				bManInterlockLiftOut := NOT bManualZIsSafe;
				bManInterlockOut := NOT ((aTRobotAxis[LA_Z1].lrCurrentPos < (alrSafePos[LA_Z1]+lrSafeTolerance)) AND (aTRobotAxis[LA_Z2].lrCurrentPos < (alrSafePos[LA_Z2]+lrSafeTolerance)) AND
								 (*(aTRobotAxis[LA_X].lrCurrentPos < (alrSafePos[LA_X]+lrSafeTolerance)) AND (aTRobotAxis[LA_Y].lrCurrentPos < (alrSafePos[LA_Y]+lrSafeTolerance)) AND*)
								(*AND ((aTRobotAxis[LA_Z1].eCurrentState = AS_InPosition) OR (aTRobotAxis[LA_Z1].eCurrentState = AS_PowerOff))
								AND ((aTRobotAxis[LA_Z2].eCurrentState = AS_InPosition)  OR (aTRobotAxis[LA_Z2].eCurrentState = AS_PowerOff))*)
								(*(aTRobotAxis[LA_X].bAxisHomed) AND (aTRobotAxis[LA_Y].bAxisHomed) AND*)
								(aTRobotAxis[LA_Z1].bAxisHomed) AND (aTRobotAxis[LA_Z2].bAxisHomed) AND bPlateTakerIsUp);
				CASE sCurrentState.eStep OF
					SP_ManualStp0 :
						TManualCmd.TPlateVacuum.Enable := TRUE;
						TManualCmd.THead1Vacuum.Enable := TRUE;
						TManualCmd.THead2Vacuum.Enable := TRUE;
						TManualCmd.TPlateVacuum.Activate := bEnablePlateVacuum;
						TManualCmd.TMovePlateTakerDown.Activate := bMovePlateTakerDown;
						TManualCmd.THead1Vacuum.Activate := abEnableHeadVacuum[0];
						TManualCmd.THead2Vacuum.Activate := abEnableHeadVacuum[1];
						FOR iAxis := 0 TO 4 DO
							TManualCmd.aTAxis[iAxis].Home.Activate := FALSE;
							TManualCmd.aTAxis[iAxis].MoveFw.Activate := FALSE;
							TManualCmd.aTAxis[iAxis].MoveBw.Activate := FALSE;
							TManualCmd.aTAxisPos[iAxis].MoveToTeach.Activate := FALSE;
							TManualCmd.aTAxisPos[iAxis].Teach := FALSE;
							TManualCmd.aTAxisPos[iAxis].MoveToTeach.Enable := FALSE;
							TManualCmd.aTAxis[iAxis].JogStep := alrJogStep[iAxis];
						END_FOR
						FOR i:= 0 TO 1 DO
							TManualCmd.alrVaccumThershold[i] := alrVacuumThreshold[i];
						END_FOR
						TManualCmd.TVisionCalibration.Activate := FALSE;
						TManualCmd.TSafe.Activate := FALSE;
						TManualCmd.TZSensorTeach.Activate := FALSE;
						 iManMoveAxis:=iManMoveAxisNone;
						TManualCmd.TAspirationBrush.Enable := TRUE;
						TManualCmd.TAspirationBrush.Activate := bAspirationBrushOn;
						TManualCmd.lrSensorAdjust := lrSensorAdjust;
						TManualCmd.TMoveVision2Table.Activate := FALSE;
						TManualCmd.TMoveVision2Lift.Activate := FALSE;
						sCurrentState.eStep := SP_ManualStp1;
					SP_ManualStp1 :
						IF bStopReq THEN
							sCurrentState.eStatus := MS_Stopped;
						ELSE
							FOR iAxis := 0 TO 4 DO
								iTeachedAxis := GetLoaderTeachedAxisFromAxis(iAxis);
								IF TManualCmd.aTAxisPos[iAxis].Teach THEN
									TManualCmd.aTAxisPos[iAxis].Teach := FALSE; (* change here the learning teach *)
									IF (iRobotOffset = LTO_Z1) THEN
										alrRobotOffset[iTeachedAxis,iRobotOffset] := 0;
										alrRobotPos[iTeachedAxis, iRobotPosition] := aTRobotAxis[iAxis].lrCurrentPos;
										iTeachedModeDebug := 0;
									ELSIF (iRobotOffset <> LTO_Plate) THEN (* Plate position are hardcoded, cannot be teached *)
										alrRobotOffset[iTeachedAxis, iRobotOffset] := aTRobotAxis[iAxis].lrCurrentPos - alrRobotPos[iTeachedAxis, iRobotPosition];
										iTeachedModeDebug := 1;
									END_IF
								END_IF
								IF (alrJogStep[iAxis] <> TManualCmd.aTAxis[iAxis].JogStep) THEN
									alrJogStep[iAxis] := TManualCmd.aTAxis[iAxis].JogStep;
								END_IF
								IF TManualCmd.aTAxisPos[iAxis].MoveToTeach.Activate AND iManMoveAxis=iManMoveAxisNone THEN
									alrTargetPos[iAxis] := TManualCmd.aTAxisPos[iAxis].TeachedPos;
									iManMoveAxis := iAxis;
									sCurrentState.eStep := SP_ManualStp10;
								END_IF
								IF TManualCmd.aTAxis[iAxis].MoveFw.Activate AND iManMoveAxis=iManMoveAxisNone THEN
									alrTargetPos[iAxis] := aTRobotAxis[iAxis].lrCurrentPos + alrJogStep[iAxis];
									iManMoveAxis := iAxis;
									sCurrentState.eStep := SP_ManualStp10;
								END_IF
								IF TManualCmd.aTAxis[iAxis].MoveBw.Activate AND iManMoveAxis=iManMoveAxisNone THEN
									alrTargetPos[iAxis] := aTRobotAxis[iAxis].lrCurrentPos - alrJogStep[iAxis];
									iManMoveAxis := iAxis;
									sCurrentState.eStep := SP_ManualStp10;
								END_IF
								IF TManualCmd.aTAxis[iAxis].Home.Activate AND  iManMoveAxis=iManMoveAxisNone THEN
									iManMoveAxis := iAxis;
									sCurrentState.eStep := SP_ManualStp20;
								END_IF
							END_FOR
							FOR i:= 0 TO 1 DO
								IF TManualCmd.alrVaccumThershold[i] <> alrVacuumThreshold[i] THEN
									alrVacuumThreshold[i] := TManualCmd.alrVaccumThershold[i];
								END_IF
							END_FOR
							IF TManualCmd.TSafe.Activate AND  iManMoveAxis=iManMoveAxisNone THEN
								TManualCmd.TSafe.Activate := FALSE;
								iManMoveAxis:=LA_X;
								sCurrentState.eStep := SP_ManualStp30;
							END_IF
							IF TManualCmd.TVisionCalibration.Activate AND  iManMoveAxis=iManMoveAxisNone THEN
								TManualCmd.TVisionCalibration.Activate := FALSE;
								iManMoveAxis:=LA_X;
								sCurrentState.eStep := SP_ManualStp50;
							END_IF
							IF (lrSensorAdjust <> TManualCmd.lrSensorAdjust) THEN
								lrSensorAdjust :=  TManualCmd.lrSensorAdjust;
							END_IF
							IF TManualCmd.TZSensorTeach.Activate THEN
								TManualCmd.TZSensorTeach.Activate := FALSE;
								lrSensorAdjust := 0 - (TSensorMeasure.lrValue - lrSensorAdjust);
								TManualCmd.lrSensorAdjust := lrSensorAdjust;
							END_IF
							IF TManualCmd.TMoveVision2Table.Activate  AND  iManMoveAxis=iManMoveAxisNone THEN
								TManualCmd.TMoveVision2Table.Activate := FALSE;
								iManMoveAxis:=LA_X;
								alrTargetPos[LA_X] := alrRobotPos[LTA_X,LTP_TableSideALayering1]  -  sPartDataMMI.alrPartOffsetLayering[sRunData.iLayringOffsetPos].lrX + alrRobotOffset[LTA_X, LTO_Vision];
								alrTargetPos[LA_Y] :=  alrRobotPos[LTA_Y,LTP_TableSideALayering1]  + sPartDataMMI.alrPartOffsetLayering[sRunData.iLayringOffsetPos].lrY + alrRobotOffset[LTA_Y, LTO_Vision];
								sCurrentState.eStep := SP_ManualStp70;
							END_IF
							IF TManualCmd.TMoveVision2Lift.Activate  AND  iManMoveAxis=iManMoveAxisNone THEN
								TManualCmd.TMoveVision2Lift.Activate := FALSE;
								iManMoveAxis:=LA_X;
								alrTargetPos[LA_X] := alrRobotPos[LTA_X,LTP_Lift1] + alrRobotOffset[LTA_X, LTO_Vision] + alrLiftCalibrationOffset[LTP_Lift1,LTA_X]  - sPlateData.alrPartOnPlate[TManualCmd.wMoveVision2LiftPos-1].lrX ;
								alrTargetPos[LA_Y] :=  alrRobotPos[LTA_Y,LTP_Lift1] + alrRobotOffset[LTA_Y, LTO_Vision] + alrLiftCalibrationOffset[LTP_Lift1,LTA_Y] - sPlateData.alrPartOnPlate[TManualCmd.wMoveVision2LiftPos-1].lrY ;
								sCurrentState.eStep := SP_ManualStp70;
							END_IF
						END_IF
					SP_ManualStp10: (* Do the movement *)
						aeMoveRobotCommand[iManMoveAxis] := AC_MoveAtAbsPos;
						sCurrentState.eStep := SP_ManualStp11;
					SP_ManualStp11: (* Wait until position is reached *)
						CASE aTRobotAxis[iManMoveAxis].eCurrentState OF
							AS_InPosition, AS_InError:
								FOR iAxis := 0 TO 4 DO
									TManualCmd.aTAxis[iAxis].Home.Activate := FALSE;
									TManualCmd.aTAxis[iAxis].MoveFw.Activate := FALSE;
									TManualCmd.aTAxis[iAxis].MoveBw.Activate := FALSE;
									TManualCmd.aTAxisPos[iAxis].MoveToTeach.Activate := FALSE;
								END_FOR
								 iManMoveAxis:=iManMoveAxisNone;
								sCurrentState.eStep := SP_ManualStp1;
						END_CASE
					SP_ManualStp20 : (* Init axis *)
						aeMoveRobotCommand[iManMoveAxis] := AC_Home;
						sCurrentState.eStep := SP_ManualStp21;
					SP_ManualStp21 : (* Rotate the turn over to go to index position *)
						CASE aTRobotAxis[iManMoveAxis].eCurrentState OF
							AS_InPosition, AS_InError:
								FOR iAxis := 0 TO 4 DO
									TManualCmd.aTAxis[iAxis].Home.Activate := FALSE;
									TManualCmd.aTAxis[iAxis].MoveFw.Activate := FALSE;
									TManualCmd.aTAxis[iAxis].MoveBw.Activate := FALSE;
								END_FOR
								 iManMoveAxis:=iManMoveAxisNone;
								sCurrentState.eStep := SP_ManualStp1;
						END_CASE
					SP_ManualStp30: (* Move taker up *)
						TManualCmd.TMovePlateTakerDown.Activate := FALSE;
						IF bPlateTakerIsUp THEN
							sCurrentState.eStep := SP_ManualStp31;
						ELSIF bJackError THEN
							iManMoveAxis:=iManMoveAxisNone;
							sCurrentState.eStep := SP_ManualStp1;
						END_IF
					SP_ManualStp31: (*Move  Z1 and Z2 to Limit*)
						aeMoveRobotCommand[LA_Z1] := AC_MoveLimitNeg;
						aeMoveRobotCommand[LA_Z2] := AC_MoveLimitNeg;
						sCurrentState.eStep := SP_ManualStp32;
					SP_ManualStp32:
						IF aTRobotAxis[LA_Z1].eCurrentState= AS_OnLimitNeg AND aTRobotAxis[LA_Z2].eCurrentState= AS_OnLimitNeg THEN
							sCurrentState.eStep := SP_ManualStp33;
						ELSIF (aTRobotAxis[LA_Z1].eCurrentState= AS_OnLimitNeg AND aTRobotAxis[LA_Z2].eCurrentState = AS_InError) OR
							    (aTRobotAxis[LA_Z1].eCurrentState= AS_InError AND aTRobotAxis[LA_Z2].eCurrentState = AS_OnLimitNeg) OR
							    (aTRobotAxis[LA_Z1].eCurrentState= AS_InError AND aTRobotAxis[LA_Z2].eCurrentState = AS_InError) THEN
							iManMoveAxis:=iManMoveAxisNone;
							sCurrentState.eStep := SP_ManualStp1;
						END_IF
					SP_ManualStp33: (* Init X/Y  *)
						aeMoveRobotCommand[LA_X] := AC_Init;
						aeMoveRobotCommand[LA_Y] := AC_Init;
						sCurrentState.eStep := SP_ManualStp34;
					SP_ManualStp34:
						IF aTRobotAxis[LA_X].eCurrentState= AS_InPosition AND aTRobotAxis[LA_Y].eCurrentState = AS_InPosition THEN
							sCurrentState.eStep := SP_ManualStp35;
						ELSIF (aTRobotAxis[LA_X].eCurrentState= AS_InPosition AND aTRobotAxis[LA_Y].eCurrentState = AS_InError) OR
							    (aTRobotAxis[LA_X].eCurrentState= AS_InError AND aTRobotAxis[LA_Y].eCurrentState = AS_InPosition) OR
							    (aTRobotAxis[LA_X].eCurrentState= AS_InError AND aTRobotAxis[LA_Y].eCurrentState = AS_InError) THEN
							iManMoveAxis:=iManMoveAxisNone;
							sCurrentState.eStep := SP_ManualStp1;
						END_IF
					SP_ManualStp35: (* Move X/Y *)
						aeMoveRobotCommand[LA_X] := AC_MoveAtAbsPos;
						aeMoveRobotCommand[LA_Y] := AC_MoveAtAbsPos;
						alrTargetPos[LA_X] := alrSafePos[LA_X];
						alrTargetPos[LA_Y] := alrSafePos[LA_Y];
						sCurrentState.eStep := SP_ManualStp36;
					SP_ManualStp36:
						IF aTRobotAxis[LA_X].eCurrentState= AS_InPosition AND aTRobotAxis[LA_Y].eCurrentState = AS_InPosition THEN
							sCurrentState.eStep := SP_ManualStp37;
						ELSIF (aTRobotAxis[LA_X].eCurrentState= AS_InPosition AND aTRobotAxis[LA_Y].eCurrentState = AS_InError) OR
							    (aTRobotAxis[LA_X].eCurrentState= AS_InError AND aTRobotAxis[LA_Y].eCurrentState = AS_InPosition) OR
							    (aTRobotAxis[LA_X].eCurrentState= AS_InError AND aTRobotAxis[LA_Y].eCurrentState = AS_InError) THEN
							iManMoveAxis:=iManMoveAxisNone;
							sCurrentState.eStep := SP_ManualStp1;
						END_IF
					SP_ManualStp37: (* Init Z1 and Z2*)
						aeMoveRobotCommand[LA_Z1] := AC_Init;
						aeMoveRobotCommand[LA_Z2] := AC_Init;
						sCurrentState.eStep := SP_ManualStp38;
					SP_ManualStp38:
						IF aTRobotAxis[LA_Z1].eCurrentState= AS_InPosition AND aTRobotAxis[LA_Z2].eCurrentState = AS_InPosition THEN
							sCurrentState.eStep := SP_ManualStp39;
						ELSIF (aTRobotAxis[LA_Z1].eCurrentState= AS_InPosition AND aTRobotAxis[LA_Z2].eCurrentState = AS_InError) OR
							    (aTRobotAxis[LA_Z1].eCurrentState= AS_InError AND aTRobotAxis[LA_Z2].eCurrentState = AS_InPosition) OR
							    (aTRobotAxis[LA_Z1].eCurrentState= AS_InError AND aTRobotAxis[LA_Z2].eCurrentState = AS_InError) THEN
							iManMoveAxis:=iManMoveAxisNone;
							sCurrentState.eStep := SP_ManualStp1;
						END_IF
					SP_ManualStp39: (* Move up Z1 and Z2 *)
						aeMoveRobotCommand[LA_Z1] := AC_MoveAtAbsPos;
						aeMoveRobotCommand[LA_Z2] := AC_MoveAtAbsPos;
						alrTargetPos[LA_Z1] := alrSafePos[LA_Z1];
						alrTargetPos[LA_Z2] := alrSafePos[LA_Z2];
						sCurrentState.eStep := SP_ManualStp40;
					SP_ManualStp40:
						IF (aTRobotAxis[LA_Z1].eCurrentState= AS_InPosition OR aTRobotAxis[LA_Z1].eCurrentState = AS_InError) AND
							    (aTRobotAxis[LA_Z2].eCurrentState= AS_InPosition OR aTRobotAxis[LA_Z2].eCurrentState = AS_InError) THEN
							iManMoveAxis:=iManMoveAxisNone;
							sCurrentState.eStep := SP_ManualStp1;
						END_IF
					SP_ManualStp50: (*Switch part for learning vision *)
						iHead := 0;
						alrTargetPos[LA_X] := alrRobotPos[LTA_X,LTP_TableSideALayering1] + alrRobotOffset[LTA_X, iHead];
						alrTargetPos[LA_Y] :=  alrRobotPos[LTA_Y,LTP_TableSideALayering1] + alrRobotOffset[LTA_Y, iHead];
						alrTargetPos[LA_THETA] := alrRobotPos[LTA_THETA,LTP_TableSideALayering1] + alrRobotOffset[LTA_THETA, iHead];
						ZPositionTakeGive := alrRobotPos[LTA_Z,LTP_TableSideALayering1] + alrRobotOffset[LTA_Z, iHead];
						alrTargetPos[LA_X] := alrTargetPos[LA_X]   -  sPartDataMMI.alrPartOffsetLayering[0].lrX;
						alrTargetPos[LA_Y] := alrTargetPos[LA_Y]  + sPartDataMMI.alrPartOffsetLayering[0].lrY;
						ZPositionTakeGive := ZPositionTakeGive + (lrCalibrationLayeringAndPartAndHeadHeight - sPartDataMMI.lrLayeringAndPartAndHeadHeight);
						aeMoveRobotCommand[LA_X] := AC_MoveAtAbsPos;
						aeMoveRobotCommand[LA_Y] := AC_MoveAtAbsPos;
						aeMoveRobotCommand[LA_THETA] := AC_MoveAtAbsPos;
						sCurrentState.eStep := SP_ManualStp51;
					SP_ManualStp51:
						IF eRobotXYTStatus = AS_InPosition THEN
							sCurrentState.eStep := SP_ManualStp52;
						END_IF
					SP_ManualStp52 :  (*Take Part*)
						ZPosition := ZPositionTakeGive + sPartDataMMI.lrPartOffsetZLayeringTake;
						alrTargetPos[LA_Z1+iHead] := ZPosition;
						aeMoveRobotCommand[LA_Z1+iHead] := AC_MoveAtAbsPos;
						sCurrentState.eStep := SP_ManualStp53;
					SP_ManualStp53 :  (*Movement done*)
						IF aTRobotAxis[LA_Z1+iHead].lrRemainingTimeToGo < 1 AND aTRobotAxis[LA_Z1+iHead].lrRemainingTimeToGo <> 0 THEN
							 TManualCmd.THead1Vacuum.Activate := TRUE;
						END_IF
						IF aTRobotAxis[LA_Z1+iHead].eCurrentState = AS_InPosition THEN
							 TManualCmd.THead1Vacuum.Activate := TRUE;
							sCurrentState.eStep := SP_ManualStp54;
						END_IF
					SP_ManualStp54 :
						(* Check if the part is on head *)
						IF aTHeadVacuum[iHead].bVacuumCorrect THEN
							alrTargetPos[LA_Z1+iHead] := alrSafePos[LA_Z1+iHead];
							aeMoveRobotCommand[LA_Z1+iHead] := AC_MoveAtAbsPos;
							sCurrentState.eStep := SP_ManualStp55;
						END_IF
					SP_ManualStp55 :  (*Movement done*)
						IF aTRobotAxis[LA_Z1+iHead].eCurrentState = AS_InPosition THEN
							iPlatePos := 0;
							iZSensorPositionScan := 0;
							sCurrentState.eStep := SP_ManualStp56;
						END_IF
					SP_ManualStp56:
						alrTargetPos[LA_X] := alrRobotPos[LTA_X,LTP_Lift2] + alrRobotOffset[LTA_X, LTO_ZSensor] + alrLiftCalibrationOffset[LTP_Lift2,LTA_X]  -  sPlateData.alrPartOnPlate[iPlatePos].lrX - sPartDataMMI.alrSensorZOffset[iZSensorPositionScan].lrX;
						alrTargetPos[LA_Y] :=alrRobotPos[LTA_Y,LTP_Lift2] + alrRobotOffset[LTA_Y, LTO_ZSensor] + alrLiftCalibrationOffset[LTP_Lift2,LTA_Y] - sPlateData.alrPartOnPlate[iPlatePos].lrY - sPartDataMMI.alrSensorZOffset[iZSensorPositionScan].lrY;
						aeMoveRobotCommand[LA_X] := AC_MoveAtAbsPos;
						aeMoveRobotCommand[LA_Y] := AC_MoveAtAbsPos;
						TSensorZWaitStab(IN := FALSE);
						sCurrentState.eStep := SP_ManualStp57;
					SP_ManualStp57:
						IF eRobotXYTStatus = AS_InPosition THEN
							TSensorZWaitStab(IN := TRUE, PT := TSensorZWaitStabTime);
							IF TSensorZWaitStab.Q THEN
								IF TSensorMeasure.bInputOutOfRange THEN
									iManMoveAxis:=iManMoveAxisNone;
									sCurrentState.eStep := SP_ManualStp1;
									bZSensorOutOfRangeError := TRUE;
								END_IF
								lrZSensorPosition[iZSensorPositionScan] := TSensorMeasure.lrValue;
								IF iZSensorPositionScan = 0 AND (sPartDataMMI.alrSensorZOffset[1].lrX<>0 OR sPartDataMMI.alrSensorZOffset[1].lrY<>0) THEN
									iZSensorPositionScan := iZSensorPositionScan + 1;
									sCurrentState.eStep := SP_ManualStp56;
								ELSE
									sCurrentState.eStep := SP_ManualStp58;
								END_IF
							END_IF
						END_IF
					SP_ManualStp58: (* Move to take position *)
						IF iZSensorPositionScan = 1 THEN
							(* We used two position, mean the value *)
							ZPositionTakeGive := (lrZSensorPosition[0] + lrZSensorPosition[1]) / 2;
						ELSE
							(* Only one position, use the first one then *)
							ZPositionTakeGive := lrZSensorPosition[0];
						END_IF
						ZPositionTakeGive := alrRobotPos[LTA_Z,LTP_TableSideALayering1] + alrRobotOffset[LTA_Z, iHead] + (lrCalibrationPartAndHeadHeight - sPartDataMMI.lrPartAndHeadHeight) - ZPositionTakeGive;
						alrTargetPos[LA_X] := alrRobotPos[LTA_X,LTP_Lift2] + alrRobotOffset[LTA_X, iHead] + alrLiftCalibrationOffset[LTP_Lift2,LTA_X]  -  sPlateData.alrPartOnPlate[iPlatePos].lrX;
						alrTargetPos[LA_Y] :=alrRobotPos[LTA_Y,LTP_Lift2] + alrRobotOffset[LTA_Y, iHead] + alrLiftCalibrationOffset[LTP_Lift2,LTA_Y] - sPlateData.alrPartOnPlate[iPlatePos].lrY;
						alrTargetPos[LA_THETA] := alrRobotPos[LTA_THETA,LTP_TableSideALayering1] + alrRobotOffset[LTA_THETA, iHead];
						aeMoveRobotCommand[LA_THETA] := AC_MoveAtAbsPos;
						aeMoveRobotCommand[LA_X] := AC_MoveAtAbsPos;
						aeMoveRobotCommand[LA_Y] := AC_MoveAtAbsPos;
						sCurrentState.eStep := SP_ManualStp59;
					SP_ManualStp59:
						IF eRobotXYTStatus = AS_InPosition THEN
							ZPosition := ZPositionTakeGive + sPartDataMMI.lrPartOffsetZLiftDrop;
							sCurrentState.eStep := SP_ManualStp60;
						END_IF
					SP_ManualStp60 : (*Give Part*)
						alrTargetPos[LA_Z1+iHead] := ZPosition + 1;
						aeMoveRobotCommand[LA_Z1+iHead] := AC_MoveAtAbsPos;
						sCurrentState.eStep := SP_ManualStp61;
					SP_ManualStp61 :  (*Movement done*)
						IF aTRobotAxis[LA_Z1+iHead].eCurrentState = AS_InPosition THEN
							 TManualCmd.THead1Vacuum.Activate := FALSE;
							sCurrentState.eStep := SP_ManualStp62;
						END_IF
					SP_ManualStp62:
						(* Check if laying vacuum is disabled *)
						IF aTHeadVacuum[iHead].bVacuumCorrect THEN
							alrTargetPos[LA_Z1+iHead] := alrSafePos[LA_Z1+iHead];
							aeMoveRobotCommand[LA_Z1+iHead] := AC_MoveAtAbsPos;
							sCurrentState.eStep := SP_ManualStp63;
						END_IF
					SP_ManualStp63 :
						IF aTRobotAxis[LA_Z1+iHead].eCurrentState = AS_InPosition THEN
							alrTargetPos[LA_X] := alrRobotPos[LTA_X,LTP_Lift2] + alrRobotOffset[LTA_X, LTO_Vision] + alrLiftCalibrationOffset[LTP_Lift2,LTA_X]  - sPlateData.alrPartOnPlate[iPlatePos].lrX ;
							alrTargetPos[LA_Y] :=  alrRobotPos[LTA_Y,LTP_Lift2] + alrRobotOffset[LTA_Y, LTO_Vision] + alrLiftCalibrationOffset[LTP_Lift2,LTA_Y] - sPlateData.alrPartOnPlate[iPlatePos].lrY ;
							aeMoveRobotCommand[LA_X] := AC_MoveAtAbsPos;
							aeMoveRobotCommand[LA_Y] := AC_MoveAtAbsPos;
							sCurrentState.eStep := SP_ManualStp64;
						END_IF
					SP_ManualStp64:
						IF eRobotXYTStatus = AS_InPosition THEN
							iManMoveAxis:=iManMoveAxisNone;
							sCurrentState.eStep := SP_ManualStp1;
						END_IF
					SP_ManualStp70: (* Move X/Y *)
						aeMoveRobotCommand[LA_X] := AC_MoveAtAbsPos;
						aeMoveRobotCommand[LA_Y] := AC_MoveAtAbsPos;
						sCurrentState.eStep := SP_ManualStp71;
					SP_ManualStp71:
						IF aTRobotAxis[LA_X].eCurrentState= AS_InPosition AND aTRobotAxis[LA_Y].eCurrentState = AS_InPosition THEN
							iManMoveAxis:=iManMoveAxisNone;
							sCurrentState.eStep := SP_ManualStp1;
						END_IF
				END_CASE
				abEnableHeadVacuum[0] := TManualCmd.THead1Vacuum.Activate;
				abEnableHeadVacuum[1] := TManualCmd.THead2Vacuum.Activate;
				bMovePlateTakerDown := TManualCmd.TMovePlateTakerDown.Activate;
				bEnablePlateVacuum := TManualCmd.TPlateVacuum.Activate;
				TManualCmd.lrSensorAdjust := lrSensorAdjust;
				bAspirationBrushOn := TManualCmd.TAspirationBrush.Activate;
			MS_Paused:
				IF bStopReq THEN
					sCurrentState.eStatus := MS_Ready;
				END_IF
		END_CASE;
	MC_Init :
		sCurrentState.eStep := SP_InitStp1;
		sCurrentState.eStatus := MS_Init;
	MC_Run :
		sCurrentState.eStatus := MS_Running;
	MC_Manual :
		sCurrentState.bInitDone := FALSE;
		sCurrentState.eStatus := MS_Manual;
		sCurrentState.eStep := SP_ManualStp0;
	MC_Stop :
		sCurrentState.eStatus := MS_Stopped;
END_CASE;

IF bResetErrors THEN
	sCurrentState.bInError := FALSE;
	bZSensorOutOfRangeError := FALSE;
END_IF

IF bNewJob THEN
	IF C_PROD_MODE_GOOD_PART THEN
		IF sProdLot.dGoodQty > 0 THEN
			sProdLot.dEstimatedPartTime := TIME_TO_DWORD(TJobElapsed)  / sProdLot.dGoodQty;
		ELSE
			sProdLot.dEstimatedPartTime := 0;
		END_IF
	ELSE
		IF sProdLot.dProdQty > 0 THEN
			sProdLot.dEstimatedPartTime := TIME_TO_DWORD(TJobElapsed)  / sProdLot.dProdQty;
		ELSE
			sProdLot.dEstimatedPartTime := 0;
		END_IF
	END_IF
	sProdLot.dLoadedQty := sProdLot.dProdQty;
END_IF

IF bNewJob THEN
(*IF bNewJob OR sCurrentState.eStatus = MS_Manual THEN*)
	abResetPlateState[LPP_Lift1] := TRUE;
	abResetPlateState[LPP_Lift2] := TRUE;
	abResetPlateState[LPP_Reject] := TRUE;
END_IF
IF bNewPlateLift1 THEN abResetPlateState[LPP_Lift1] := TRUE; END_IF
IF bNewPlateLift2 THEN abResetPlateState[LPP_Lift2] := TRUE; END_IF
IF bNewPlateReject THEN abResetPlateState[LPP_Reject] := TRUE; END_IF

IF abCopySwitchFromPlate THEN
	abCopySwitchFromPlate := FALSE;
	FOR j := 0 TO sPlateData.iNbPartOnPlate DO
		aTPartOnSwitchPlate[j].ePartStatus := aTPartOnPlate[LPP_Lift1, j].ePartStatus;
	END_FOR
END_IF

FOR i :=LPP_Reject  TO LPP_Lift2 DO
	IF abResetPlateState[i] THEN
		abResetPlateState[i] := FALSE;
		FOR j := 0 TO sPlateData.iNbPartOnPlate DO
			aTPartOnPlate[i, j ].ePartStatus := PPS_Undefined;
		END_FOR
	END_IF
END_FOR

IF abCopySwitchToPlate THEN
	abCopySwitchToPlate := FALSE;
	FOR j := 0 TO sPlateData.iNbPartOnPlate DO
		aTPartOnPlate[LPP_Lift2, j].ePartStatus := aTPartOnSwitchPlate[j].ePartStatus;
	END_FOR
END_IF
(* ----------------------------------------------------------- MOVE SECURITY CHECK -------------------------------------------------------------------------*)

(* Check if a consequent move more then 2 mm with heads down or plate taker down is requested *)
IF ((ABS(aTRobotAxis[LA_X].lrCurrentPos - alrTargetPos[LA_X]) > lrMaxXYMoveAllowed) AND (aeMoveRobotCommand[LA_X] <> AC_None)) OR
		((ABS(aTRobotAxis[LA_Y].lrCurrentPos - alrTargetPos[LA_Y]) > lrMaxXYMoveAllowed) AND (aeMoveRobotCommand[LA_Y] <> AC_None)) THEN
	IF (aTRobotAxis[LA_Z1].lrCurrentPos > (alrSecuredSafeZPos[0] + lrSafeTolerance))
			OR (aTRobotAxis[LA_Z2].lrCurrentPos > (alrSecuredSafeZPos[1] + lrSafeTolerance))
			OR NOT bPlateTakerIsUp THEN
		IF sCurrentState.eStep <> SP_RunStp63 THEN (* Do not check during cleaning *)
			aeMoveRobotCommand[LA_X] := AC_ForceStop;
			aeMoveRobotCommand[LA_Y] := AC_ForceStop;
			aeMoveRobotCommand[LA_Z1] := AC_ForceStop;
			aeMoveRobotCommand[LA_Z2] := AC_ForceStop;
			sCurrentState.bInitDone := FALSE;
			bConflictDetected := TRUE;
		END_IF
	END_IF
ELSIF ((aTRobotAxis[LA_X].lrCurrentPos > alrUnsecuredArea[0,LA_X]+ lrSafeTolerance) AND (aTRobotAxis[LA_X].lrCurrentPos < alrUnsecuredArea[1,LA_X] - lrSafeTolerance)		(* The Restritcted aera is lrSafeTolerance smaller for the axis have some space to work *)
		AND (aTRobotAxis[LA_Y].lrCurrentPos > alrUnsecuredArea[0,LA_Y]+ lrSafeTolerance) AND (aTRobotAxis[LA_Y].lrCurrentPos < alrUnsecuredArea[1,LA_Y] - lrSafeTolerance)
		AND ((aTRobotAxis[LA_Z1].lrCurrentPos > (alrSafePos[LA_Z1] + lrSafeTolerance))
		OR (aTRobotAxis[LA_Z2].lrCurrentPos > (alrSafePos[LA_Z2] + lrSafeTolerance)))) THEN
	IF (sCurrentState.eStatus = MS_Manual) OR (sCurrentState.eStatus = MS_Init) OR (sCurrentState.eStatus = MS_Stopped) THEN
		bConflictDetected := false;
	ELSE
		aeMoveRobotCommand[LA_X] := AC_ForceStop;
		aeMoveRobotCommand[LA_Y] := AC_ForceStop;
		aeMoveRobotCommand[LA_Z1] := AC_ForceStop;
		aeMoveRobotCommand[LA_Z2] := AC_ForceStop;
		sCurrentState.bInitDone := FALSE;
		bUnsecuredAeraEntry := TRUE;
		bConflictDetected := TRUE;	
	END_IF
END_IF

(* ------------------------------------------------------ END OF MOVE SECURITY CHECK -------------------------------------------------------------------*)

(* Robot command *)

IF (sCurrentState.eStatus = MS_Manual) THEN
	FOR iAxis:=0 TO 4 DO
		IF bManualZIsSafe THEN
			alrRobotSpeed[iAxis] := aTRobotAxis[iAxis].lrFastManualSpeed;
		ELSE
			alrRobotSpeed[iAxis] := aTRobotAxis[iAxis].lrManualSpeed;;
		END_IF
	END_FOR
END_IF

aTRobotAxis[LA_X](
	eCommand 		:= aeMoveRobotCommand[LA_X],
	lrTargetPos 		:= alrTargetPos[LA_X],
	lrTargetSpeed 	:= alrRobotSpeed[LA_X],
	lrAcceleration  := alrRobotAcceleration[LA_X],
	lrDeceleration	:= alrRobotDeceleration[LA_X],
	lrJerk			:= alrRobotJerk[LA_X],
	sAxis		 	:= sXAxisRef,
	bHomeSensor 	:= bHomeX,
	eAxisType		:= AT_AX5000,
	bPowerIsOn		:= bPowerOn,
	bPosLimitSwitch	:= NOT bLimitPosX,
	bNegLimitSwitch	:= NOT bLimitNegX,
	lrMoveOutDist	:= 100,
	bResetErrors	 	:= bResetErrors,
	stServoButton 	:= TManualCmd.aTAxis[LA_X].ServoON
	);
aeMoveRobotCommand[LA_X] := AC_None;
bXAxisError := (aTRobotAxis[LA_X].eCurrentState = AS_InError);

aTRobotAxis[LA_Y](
	eCommand 		:= aeMoveRobotCommand[LA_Y],
	lrTargetPos 		:= alrTargetPos[LA_Y],
	lrTargetSpeed 	:= alrRobotSpeed[LA_Y],
	lrAcceleration  := alrRobotAcceleration[LA_Y],
	lrDeceleration	:= alrRobotDeceleration[LA_Y],
	lrJerk			:= alrRobotJerk[LA_Y],
	sAxis		 	:= sYAxisRef,
	bHomeSensor 	:= bHomeY,
	eAxisType		:= AT_AX5000,
	bPowerIsOn		:= bPowerOn,
	bPosLimitSwitch	:= NOT bLimitPosY,
	bNegLimitSwitch	:= NOT bLimitNegY,
	lrMoveOutDist	:= 100,
	bResetErrors	 	:= bResetErrors,
	stServoButton 	:= TManualCmd.aTAxis[LA_Y].ServoON

);
aeMoveRobotCommand[LA_Y] := AC_None;
bYAxisError := (aTRobotAxis[LA_Y].eCurrentState = AS_InError);

aTRobotAxis[LA_Z1](
	eCommand 		:= aeMoveRobotCommand[LA_Z1],
	lrTargetPos 		:= alrTargetPos[LA_Z1],
	lrTargetSpeed 	:= alrRobotSpeed[LA_Z1],
	sAxis	 		:= sZ1AxisRef,
	bHomeSensor 	:= bHomeZ1,
	bPowerIsOn		:= bPowerOn,
	bPosLimitSwitch	:= NOT bLimitPosZ1,
	bNegLimitSwitch	:= NOT bLimitNegZ1,
	lrMoveOutDist	:= 10,
	bResetErrors	 	:= bResetErrors,
	stServoButton 	:= TManualCmd.aTAxis[LA_Z1].ServoON
);
aeMoveRobotCommand[LA_Z1] := AC_None;
bZ1AxisError := (aTRobotAxis[LA_Z1].eCurrentState = AS_InError);

aTRobotAxis[LA_Z2](
	eCommand 		:= aeMoveRobotCommand[LA_Z2],
	lrTargetPos 		:= alrTargetPos[LA_Z2],
	lrTargetSpeed 	:= alrRobotSpeed[LA_Z2],
	sAxis		 	:= sZ2AxisRef,
	bHomeSensor 	:= bHomeZ2,
	bPowerIsOn		:= bPowerOn,
	bPosLimitSwitch	:= NOT bLimitPosZ2,
	bNegLimitSwitch	:= NOT bLimitNegZ2,
	lrMoveOutDist	:= 10,
	bResetErrors	 	:= bResetErrors,
	stServoButton 	:= TManualCmd.aTAxis[LA_Z2].ServoON
);
aeMoveRobotCommand[LA_Z2] := AC_None;
bZ2AxisError := (aTRobotAxis[LA_Z2].eCurrentState = AS_InError);

aTRobotAxis[LA_THETA](
	eCommand 		:= aeMoveRobotCommand[LA_THETA],
	lrTargetPos 		:= alrTargetPos[LA_THETA],
	lrTargetSpeed 	:= alrRobotSpeed[LA_THETA],
	sAxis		 	:= sThetaAxisRef,
	bPowerIsOn		:= bPowerOn,
	bResetErrors	 	:= bResetErrors,
	eHomingAxisType := AHT_OnZeroEncoder,
	stServoButton 	:= TManualCmd.aTAxis[LA_THETA].ServoON
);
aeMoveRobotCommand[LA_THETA] := AC_None;
bTAxisError := (aTRobotAxis[LA_THETA].eCurrentState = AS_InError);

(* Get move result *)
eRobotXYTStatus := AS_Moving;
IF (aTRobotAxis[LA_X].eCurrentState = AS_InError) OR (aTRobotAxis[LA_Y].eCurrentState = AS_InError) OR (aTRobotAxis[LA_THETA].eCurrentState = AS_InError) THEN
	eRobotXYTStatus := AS_InError;
ELSIF (aTRobotAxis[LA_X].eCurrentState = AS_InPosition) AND (aTRobotAxis[LA_Y].eCurrentState = AS_InPosition) AND (aTRobotAxis[LA_THETA].eCurrentState = AS_InPosition) THEN
		eRobotXYTStatus := AS_InPosition;
END_IF

(* Handle part vacuum *)
aTHeadVacuum[0](
	bEnableVacuum		:= abEnableHeadVacuum[0],
	tVacErrorDelay		:= INT_TO_TIME(sVaccumSettingsHead.iErrorDelay),
	tBlowingTime			:= INT_TO_TIME(sVaccumSettingsHead.iBlowing),
	tWaitVacuumOK		:= INT_TO_TIME(sVaccumSettingsHead.iWaitWhenVacuumOk),
	bReset				:= bResetErrors  OR abResetVacuum[0],
	iVacuum				:= iHead1VacuumFlow,
	lrVacuumThreshold	 :=  alrVacuumThreshold[0],
	bDisableVacuumChecking := abBypassVacuumError[0],
	bVacuumOn			=> bActivateHead1Vacuum,
	bBlowOn				=> bActivateHead1Blowing,
	bVacuumError		=> bHead1VacuumError
);
abResetVacuum[0] := FALSE;
IF abBypassVacuumError[0] AND sCurrentState.eStatus = MS_Running THEN
	bHead1VacuumError := FALSE;
END_IF
IF (bResetErrors AND (sCurrentState.eStatus = MS_Stopped) AND bHead1VacuumError) THEN
	abEnableHeadVacuum[0] := FALSE;
END_IF

aTHeadVacuum[1](
	bEnableVacuum		:= abEnableHeadVacuum[1],
	tVacErrorDelay		:= INT_TO_TIME(sVaccumSettingsHead.iErrorDelay),
	tBlowingTime			:= INT_TO_TIME(sVaccumSettingsHead.iBlowing),
	tWaitVacuumOK		:= INT_TO_TIME(sVaccumSettingsHead.iWaitWhenVacuumOk),
	bReset				:= bResetErrors  OR abResetVacuum[1],
	iVacuum				:= iHead2VacuumFlow,
	lrVacuumThreshold	 :=  alrVacuumThreshold[1],
	bDisableVacuumChecking := abBypassVacuumError[1],
	bVacuumOn			=> bActivateHead2Vacuum,
	bBlowOn				=> bActivateHead2Blowing,
	bVacuumError		=> bHead2VacuumError
);
abResetVacuum[1] := FALSE;
IF abBypassVacuumError[1] AND sCurrentState.eStatus = MS_Running THEN
	bHead2VacuumError := FALSE;
END_IF
IF (bResetErrors AND (sCurrentState.eStatus = MS_Stopped) AND bHead2VacuumError) THEN
	abEnableHeadVacuum[1] := FALSE;
END_IF

(* Handle plate vacuum *)
TPlateVacuum(
	tVacErrorDelay		:= INT_TO_TIME(sVaccumSettingsPlate.iErrorDelay),
	tBlowingTime			:= INT_TO_TIME(sVaccumSettingsPlate.iBlowing),
	tWaitVacuumOK		:= INT_TO_TIME(sVaccumSettingsPlate.iWaitWhenVacuumOk),
	bEnableVacuum	:= bEnablePlateVacuum,
	bReset			:= bResetErrors,
	bVacuumOK		:= bPlateVacuumIsOk,
	bVacuumOn		=> bActivatePlateVacuum,
	bBlowOn			=> bActivatePlateBlowing,
	bVacuumError	=> bPlateVacuumError
);

(* Check jack error *)
TCheckJack(
	bJackGoOut	:= bMovePlateTakerDown,
	bJackIsIn	:= bPlateTakerIsUp,
	bJackIsOut	:= bPlateTakerIsDown,
	tTimeOut		:= t#2s,
	bResetErrors := bResetErrors,
	bJackError	=> bJackError
);

IF bJackError OR bXAxisError OR bYAxisError OR bZ1AxisError OR bZ2AxisError OR bTAxisError OR bHead1VacuumError OR bHead2VacuumError OR bPlateVacuumError OR bConflictDetected  OR bZSensorOutOfRangeError THEN
	sCurrentState.bInError := TRUE;
	IF (sCurrentState.eStatus <> MS_Manual) AND (sCurrentState.eStatus <> MS_Stopped) AND (sCurrentState.eStatus <> MS_Init) THEN
		sCurrentState.eStatus := MS_Ready;
	END_IF
END_IF

IF (NOT bPowerOn OR bXAxisError OR bYAxisError OR bZ1AxisError OR bZ2AxisError OR bTAxisError) THEN
	sCurrentState.bInitDone := FALSE;
	IF (sCurrentState.eStatus <> MS_Manual) THEN
		sCurrentState.eStatus := MS_Stopped;
	END_IF
END_IF

IF bNewJob THEN
(*	sProdLot.dProdQty := 0;
	sProdLot.dGoodQty := 0;
	sProdLot.dLoadedQty := 0; *)
	sProdLot.dEstimatedTimeLeft := 0;
END_IF
sProdLot.dProductionTime := TIME_TO_DWORD(TJobElapsed);

CASE sRunData.eModule OF
	LMP_Table:
		sOutGiveToTable := sOutGiveToModule;
		sOutTakeFromTable := sOutTakeFromModule;
	LMP_TurnOverFix,LMP_TurnOverArm:
		sOutGiveToTurnOver := sOutGiveToModule;
		sOutTakeFromTurnOver := sOutTakeFromModule;
END_CASE

(* Detect if lift seems to move to refresh Z position *)
IF eLift1RunStatus <> RS_WaitRequest THEN
	alrZLiftPos[LTP_Lift1] := 0;
END_IF
IF eLift2RunStatus <> RS_WaitRequest THEN
	alrZLiftPos[LTP_Lift2] := 0;
END_IF

sRunData.lrZPositionTakeGive := ZPositionTakeGive;
bVacuumInUse := bEnablePlateVacuum OR (abEnableHeadVacuum[0] AND NOT bHead1VacuumError)  OR (abEnableHeadVacuum[1] AND NOT bHead2VacuumError) ;
bMovePlateTakerUp := NOT bMovePlateTakerDown;

sCurrentState.bInterlocked := bManInterlock AND  (sCurrentState.eStatus = MS_Manual);
bModuleError := sCurrentState.bInError;
sCurrentState.bRunning := (sCurrentState.eStatus = MS_Running);
IF (sCurrentState.eStatus <> MS_Running) THEN eRunStatus := RS_NotRunning; END_IF

iStep := sCurrentState.eStep;

END_FUNCTION_BLOCK

(* stored: Version 1.1.0.1, ProductVersion 3.1.4022.18
   POU LoaderHdl: Id {2ccba174-361e-4ee8-a2b0-425a1f6fc94e}, SpecialFunc None *)
